// Mitsubishi GX Works2 project: Group_4   PLC: FX3G

// global labels: Global1
VAR_GLOBAL
  LightWork AT Y007 : BOOL;
  StartDay AT X007 : BOOL;
  EmergencyBut AT X011 : BOOL;
  StartCooking AT X001 : BOOL;
END_VAR
VAR_GLOBAL CONSTANT
  Lager : REAL := 5;
END_VAR
VAR_GLOBAL
  StartStockYeast AT D1101 : REAL;
  StockYeast AT D1103 : REAL;
  StartStockMalt AT D1105 : REAL;
  StockMalt AT D1107 : REAL;
  StartStockHops AT D1109 : REAL;
  StockHops AT D1111 : REAL;
END_VAR
VAR_GLOBAL CONSTANT
  MinYeast : REAL := 150;
  MinMalt : REAL := 12;
  MinHops : REAL := 60;
END_VAR
VAR_GLOBAL
  EnoughYeast AT M0 : BOOL;
  EnoughMalt AT M1 : BOOL;
  EnoughHops AT M2 : BOOL;
END_VAR
VAR_GLOBAL CONSTANT
  Pilzner : REAL := 6;
  MinYeastP : REAL := 150;
  MinYeastL : REAL := 150;
  MinMaltL : REAL := 12;
  MinMaltP : REAL := 6;
  MinHopsP : REAL := 53;
  MinHopsL : REAL := 60;
END_VAR
VAR_GLOBAL
  Y1Controler AT M3 : BOOL;
  CookingTime AT Y001 : BOOL;
  cook AT TC19 : BOOL;
END_VAR
VAR_GLOBAL CONSTANT
  CookDest : INT := 40;
END_VAR
VAR_GLOBAL
  cookFinish AT TS19 : BOOL;
  LagerBulb AT M10 : BOOL;
  PilznerBulb AT M11 : BOOL;
  HelpM12 AT M12 : BOOL;
  HelpLight AT M12 : BOOL;
  HelpLight10 AT M12 : BOOL;
  HelpLight11 AT M12 : BOOL;
  AnalogAsFloat AT D1221 : REAL;
END_VAR
VAR_GLOBAL CONSTANT
  Divider : REAL := 400;
END_VAR
VAR_GLOBAL
  AnalogInput1 AT D8280 : INT;
  SaveAnalog1 AT D8201 : INT;
  cookTimerAnswer AT TS19 : BOOL;
  StartFermentation AT X005 : BOOL;
END_VAR
VAR_GLOBAL CONSTANT
  LagerFerm3Sec : INT := 30;
  PilzFerm4Sec : INT := 40;
END_VAR
VAR_GLOBAL
  FermTimer AT D1323 : INT;
  Light4 AT M4 : BOOL;
  FirstLightT21 AT TC21 : BOOL;
  Tss21 AT TS21 : BOOL;
  FirstLightAnswer AT TS21 : BOOL;
  FirstLightFerm AT Y003 : BOOL;
  SecondLightFerm AT Y004 : BOOL;
  SecondLightAnswer AT TS23 : BOOL;
  SecondLightT23 AT TC23 : BOOL;
  StartStorage AT X002 : BOOL;
  countBottle AT CC1 : BOOL;
END_VAR
VAR_GLOBAL CONSTANT
  SixBottle : INT := 6;
END_VAR
VAR_GLOBAL
  countSix AT CC2 : BOOL;
  StorageSix AT D1116 : REAL;
END_VAR
VAR_GLOBAL CONSTANT
  OneSix : REAL := 1;
END_VAR
VAR_GLOBAL
  OneBottle AT X000 : BOOL;
  FirstC1 AT CC1 : BOOL;
  LightStorage AT Y002 : BOOL;
  StorageLight AT Y002 : BOOL;
  CountFirstBottle AT CC2 : BOOL;
END_VAR
VAR_GLOBAL CONSTANT
  FirstBottle : REAL := 1;
END_VAR
VAR_GLOBAL
  FinishPacking AT M5 : BOOL;
  HelpLightM51 AT M51 : BOOL;
  checkIf5 AT TC19 : BOOL;
  HelpM20 AT M20 : BOOL;
  HelpLight18 AT M18 : BOOL;
  HelpLightM20 AT M20 : BOOL;
  HelpLightM77 AT M77 : BOOL;
  HelpLightM90 AT M90 : BOOL;
  EnoughIng AT M35 : BOOL;
  NotEnoughIng AT M35 : BOOL;
  NotEnoughYeast AT M0 : BOOL;
  NotEnoughMalt AT M1 : BOOL;
  NotEnoughHops AT M2 : BOOL;
  HelpLight60 AT M60 : BOOL;
  HelpLight61 AT M61 : BOOL;
  HelpLight62 AT M62 : BOOL;
  CookFinished AT M63 : BOOL;
  TimerLight AT M64 : BOOL;
  LightTimer AT TC25 : BOOL;
END_VAR
VAR_GLOBAL CONSTANT
  Light1 : INT := 5;
END_VAR
VAR_GLOBAL
  TimerFinished AT TS25 : BOOL;
  SixBottles AT CS1 : BOOL;
  StartCount AT M70 : BOOL;
END_VAR
VAR_GLOBAL CONSTANT
  DividerForOutput : INT := 10;
END_VAR
VAR_GLOBAL
  HowManySix AT D1136 : REAL;
  IntHowManySix AT D8002 : INT;
  OutPut AT D8282 : INT;
END_VAR
VAR_GLOBAL CONSTANT
  Constant40 : REAL := 40;
END_VAR
VAR_GLOBAL
  HelpLight81 AT M81 : BOOL;
  HelpLight80 AT M80 : BOOL;
END_VAR

// task Task_01 (event TRUE, interval 0, priority 31): POU_01

PROGRAM POU_01
(* structured ladder/FBD written out as ST: instructions are called as NAME(EN, inputs, outputs); _pN, _eN, _tN stand for wires *)
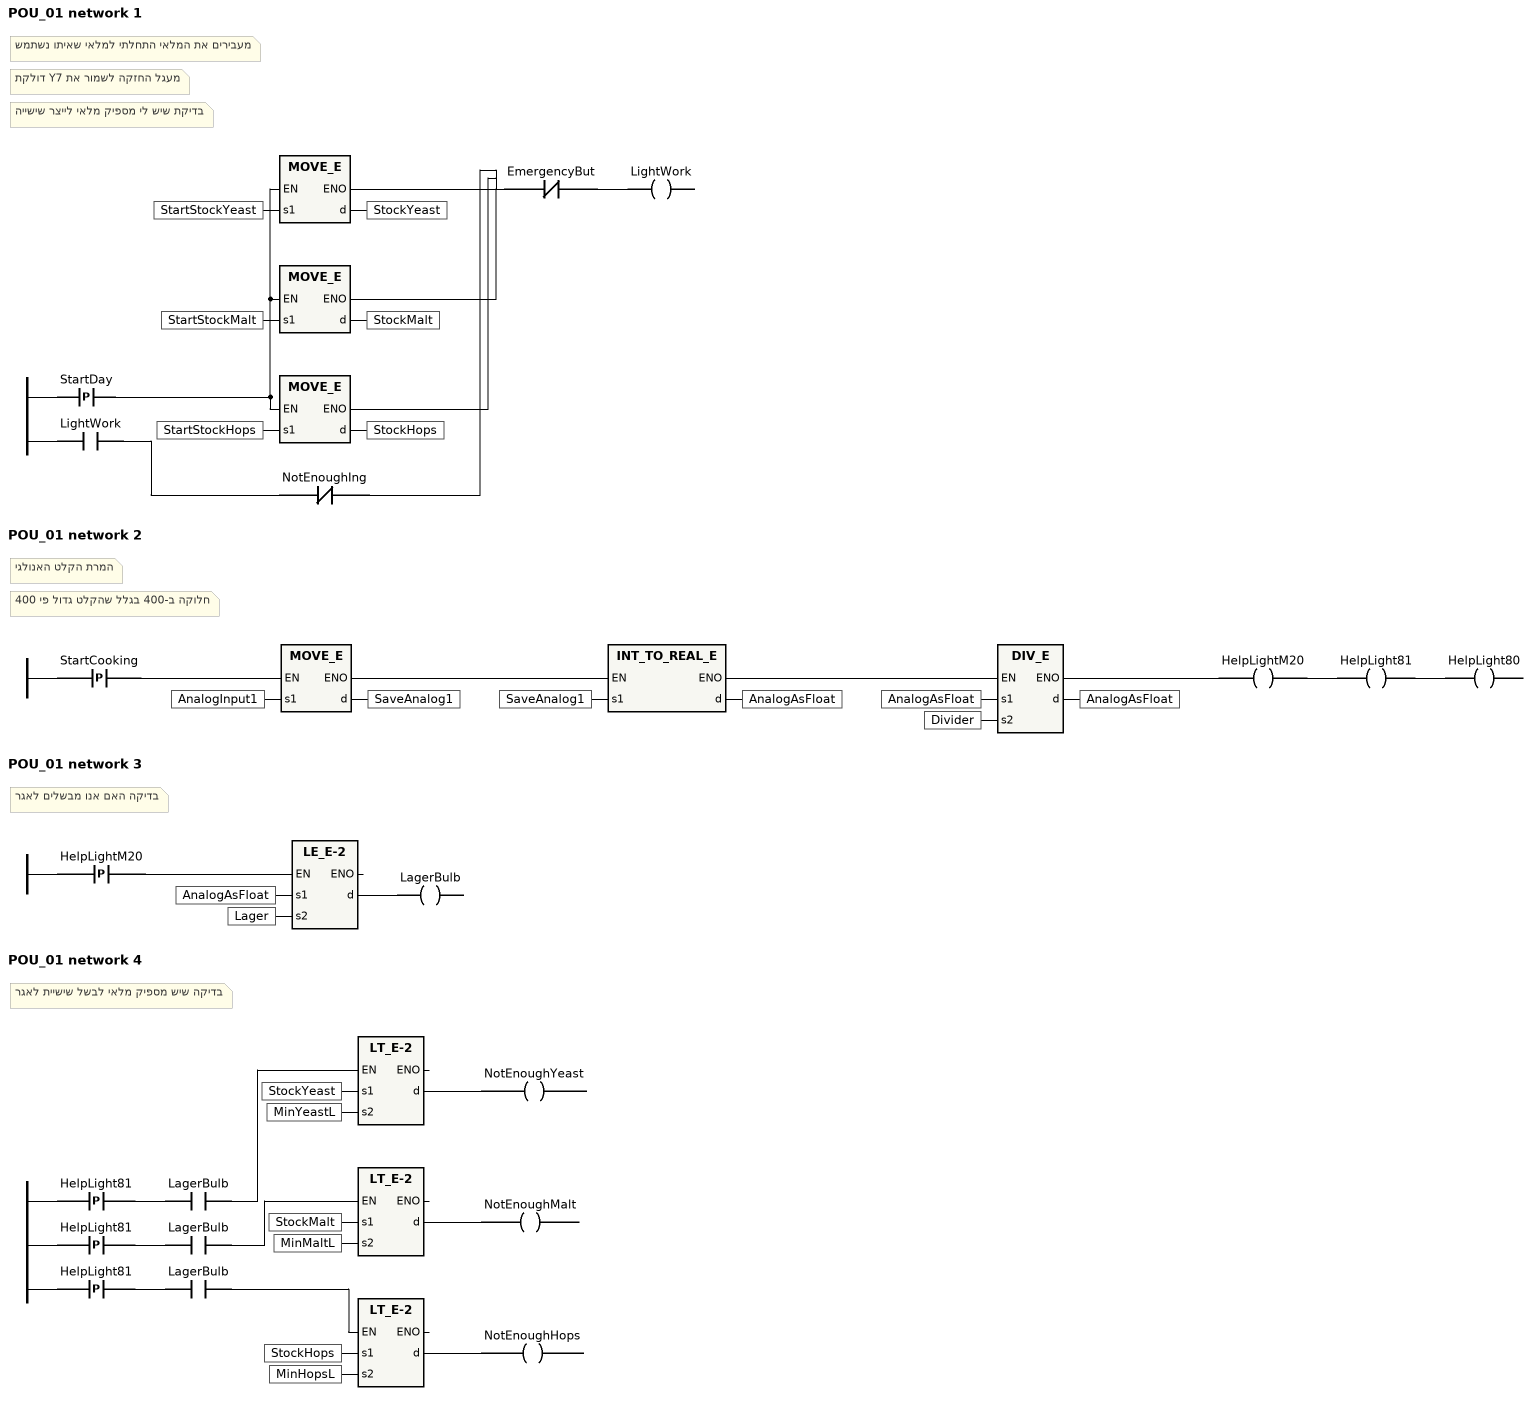
(* network 1 Day Init *)
(* מעבירים את המלאי התחלתי למלאי שאיתו נשתמש *)
(* מעגל החזקה לשמור את Y7 דולקת *)
(* בדיקת שיש לי מספיק מלאי לייצר שישייה *)
_p1 := LDP(TRUE, StartDay);
_e2 := MOVE_E(_p1, StartStockYeast, StockYeast);
_e3 := MOVE_E(_p1, StartStockMalt, StockMalt);
_e4 := MOVE_E(_p1, StartStockHops, StockHops);
LightWork := (_e2 OR _e3 OR _e4 OR (LightWork AND NOT NotEnoughIng)) AND NOT EmergencyBut;
(* network 2 StartCook *)
(* המרת הקלט האנולגי *)
(* חלוקה ב-400 בגלל שהקלט גדול פי 400 *)
_e1 := MOVE_E(LDP(TRUE, StartCooking), AnalogInput1, SaveAnalog1);
_e2 := INT_TO_REAL_E(_e1, SaveAnalog1, AnalogAsFloat);
_e3 := DIV_E(_e2, AnalogAsFloat, Divider, AnalogAsFloat);
HelpLightM20 := _e3;
HelpLight81 := _e3;
HelpLight80 := _e3;
(* network 3 CookLage *)
(* בדיקה האם אנו מבשלים לאגר *)
LE_E(LDP(TRUE, HelpLightM20), AnalogAsFloat, Lager, _t1);
LagerBulb := _t1;
(* network 4 LagCondition *)
(* בדיקה שיש מספיק מלאי לבשל שישיית לאגר *)
LT_E(LDP(TRUE, HelpLight81) AND LagerBulb, StockYeast, MinYeastL, _t1);
NotEnoughYeast := _t1;
LT_E(LDP(TRUE, HelpLight81) AND LagerBulb, StockMalt, MinMaltL, _t2);
NotEnoughMalt := _t2;
LT_E(LDP(TRUE, HelpLight81) AND LagerBulb, StockHops, MinHopsL, _t3);
NotEnoughHops := _t3;
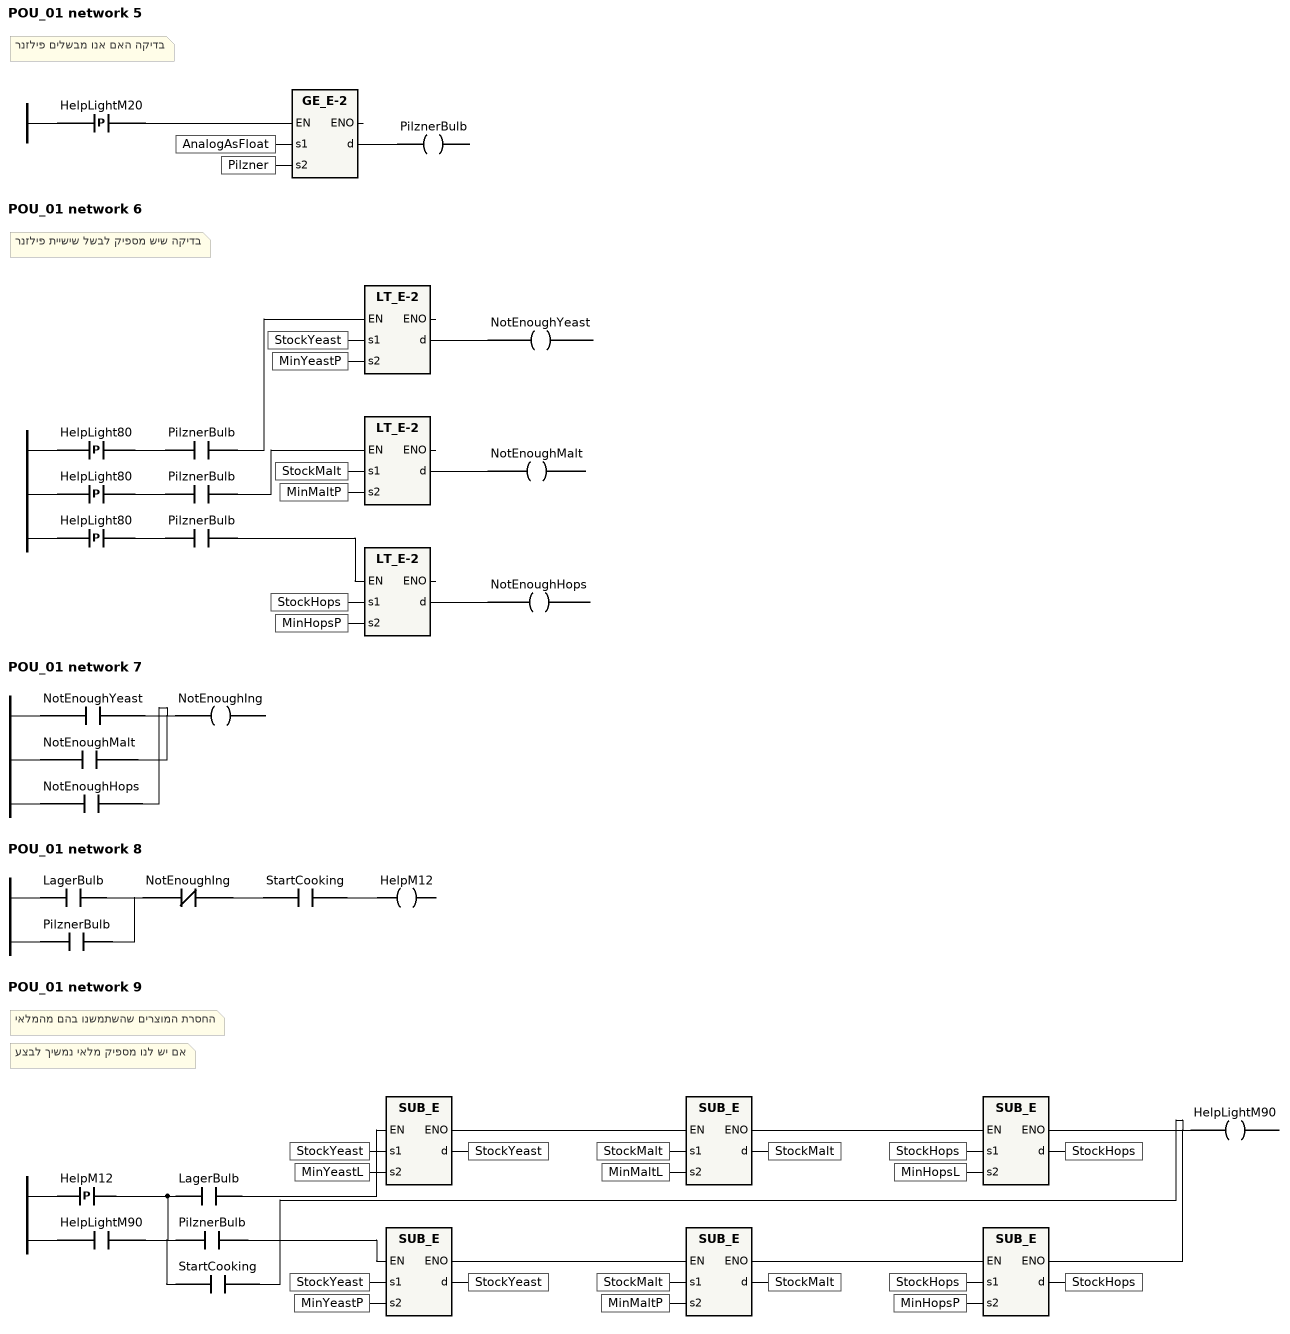
(* network 5 CookPilz *)
(* בדיקה האם אנו מבשלים פילזנר *)
GE_E(LDP(TRUE, HelpLightM20), AnalogAsFloat, Pilzner, _t1);
PilznerBulb := _t1;
(* network 6 PilzCondition *)
(* בדיקה שיש מספיק לבשל שישיית פילזנר *)
LT_E(LDP(TRUE, HelpLight80) AND PilznerBulb, StockYeast, MinYeastP, _t1);
NotEnoughYeast := _t1;
LT_E(LDP(TRUE, HelpLight80) AND PilznerBulb, StockMalt, MinMaltP, _t2);
NotEnoughMalt := _t2;
LT_E(LDP(TRUE, HelpLight80) AND PilznerBulb, StockHops, MinHopsP, _t3);
NotEnoughHops := _t3;
(* network 7 StockChecking *)
NotEnoughIng := NotEnoughYeast OR NotEnoughMalt OR NotEnoughHops;
(* network 8 CookingPermission *)
HelpM12 := ((LagerBulb OR PilznerBulb) AND NOT NotEnoughIng) AND StartCooking;
(* network 9 Cooking *)
(* החסרת המוצרים שהשתמשנו בהם מהמלאי *)
(* אם יש לנו מספיק מלאי נמשיך לבצע *)
_p1 := LDP(TRUE, HelpM12);
_e2 := SUB_E(_p1 AND LagerBulb, StockYeast, MinYeastL, StockYeast);
_e3 := SUB_E(_e2, StockMalt, MinMaltL, StockMalt);
_e4 := SUB_E(_e3, StockHops, MinHopsL, StockHops);
_e5 := SUB_E(_p1 AND PilznerBulb, StockYeast, MinYeastP, StockYeast);
_e6 := SUB_E(_e5, StockMalt, MinMaltP, StockMalt);
_e7 := SUB_E(_e6, StockHops, MinHopsP, StockHops);
HelpLightM90 := _e4 OR _e7 OR (HelpLightM90 AND StartCooking);
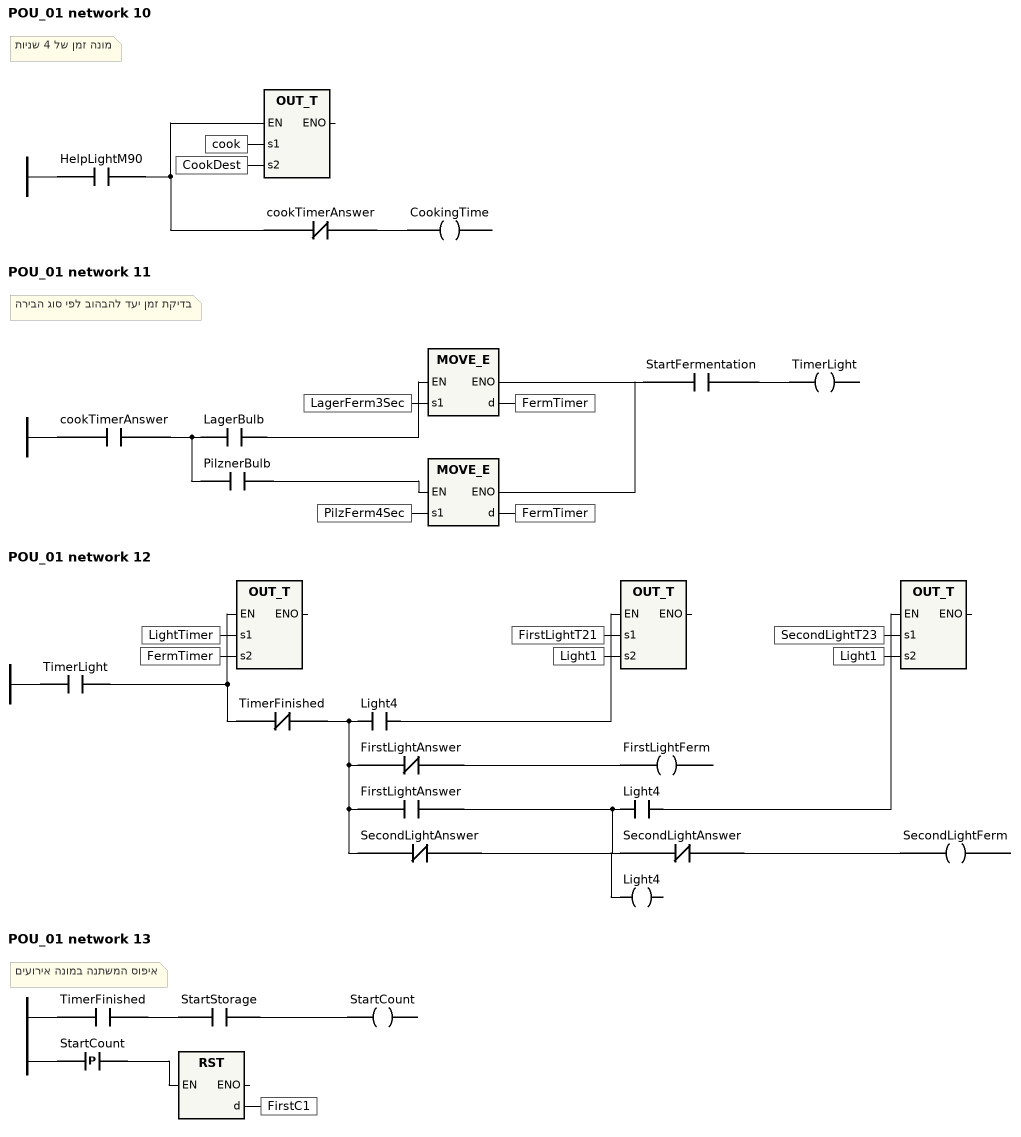
(* network 10 LightCooking *)
(* מונה זמן של 4 שניות *)
OUT_T(HelpLightM90, cook, CookDest);
CookingTime := HelpLightM90 AND NOT cookTimerAnswer;
(* network 11 Fermentation *)
(* בדיקת זמן יעד להבהוב לפי סוג הבירה *)
_e1 := MOVE_E(cookTimerAnswer AND LagerBulb, LagerFerm3Sec, FermTimer);
_e2 := MOVE_E(cookTimerAnswer AND PilznerBulb, PilzFerm4Sec, FermTimer);
TimerLight := (_e1 OR _e2) AND StartFermentation;
(* network 12 Flickering *)
OUT_T(TimerLight, LightTimer, FermTimer);
_p1 := TimerLight AND NOT TimerFinished;
OUT_T(_p1 AND Light4, FirstLightT21, Light1);
FirstLightFerm := _p1 AND NOT FirstLightAnswer;
_p2 := _p1 AND FirstLightAnswer;
OUT_T(_p2 AND Light4, SecondLightT23, Light1);
SecondLightFerm := _p2 AND NOT SecondLightAnswer;
Light4 := _p1 AND NOT SecondLightAnswer;
(* network 13 Storage *)
(* איפוס המשתנה במונה אירועים *)
StartCount := TimerFinished AND StartStorage;
RST(LDP(TRUE, StartCount), FirstC1);
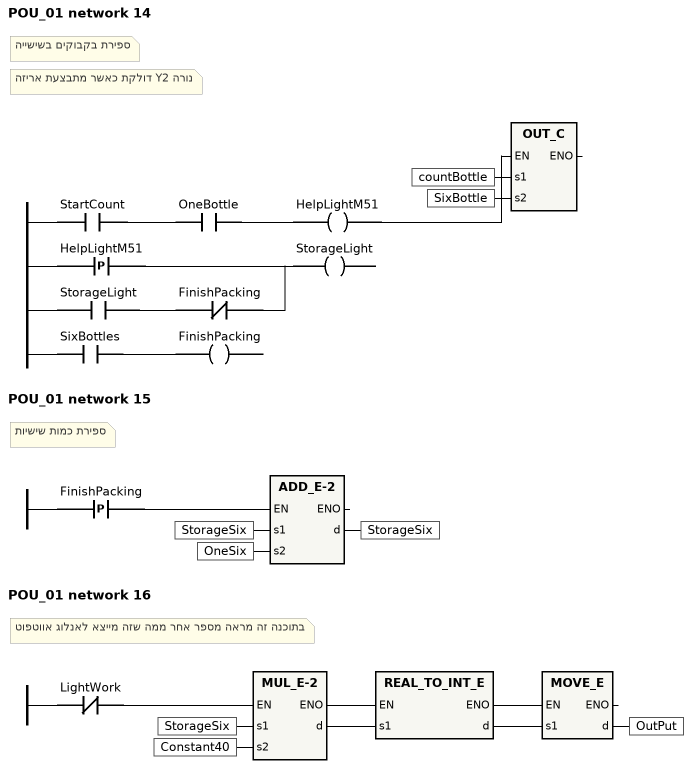
(* network 14 Packing *)
(* ספירת בקבוקים בשישייה *)
(* נורה Y2 דולקת כאשר מתבצעת אריזה *)
_p1 := StartCount AND OneBottle;
HelpLightM51 := _p1;
OUT_C(_p1, countBottle, SixBottle);
StorageLight := LDP(TRUE, HelpLightM51) OR (StorageLight AND NOT FinishPacking);
FinishPacking := SixBottles;
(* network 15 CountPackges *)
(* ספירת כמות שישיות *)
ADD_E(LDP(TRUE, FinishPacking), StorageSix, OneSix, StorageSix);
(* network 16 EndDayOutput *)
(* בתוכנה זה מראה מספר אחר ממה שזה מייצא לאנלוג אווטפוט *)
_e2 := MUL_E(NOT LightWork, StorageSix, Constant40, _t1);
_e4 := REAL_TO_INT_E(_e2, _t1, _t3);
MOVE_E(_e4, _t3, OutPut);
END_PROGRAM
